// Mitsubishi GX Works2 project: 电路控制2   PLC: FX2N/FX2NC

PROGRAM MAIN
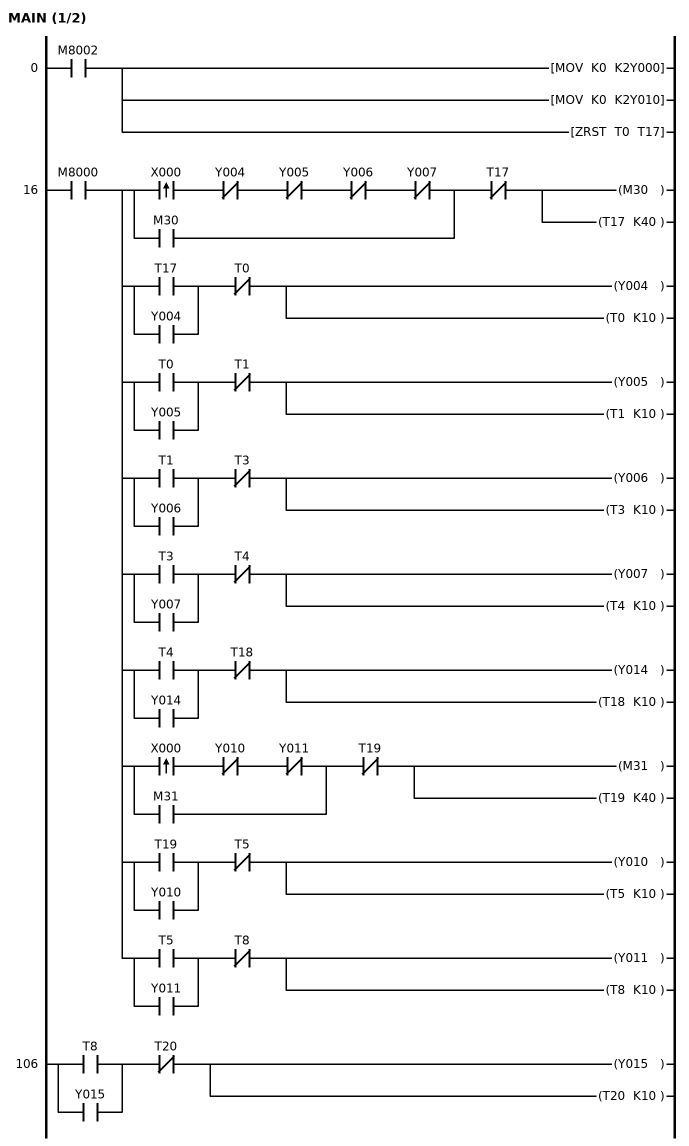
0     LD      M8002
      MOV     K0 K2Y000
      MOV     K0 K2Y010
      ZRST    T0 T17
16    LD      M8000
      MPS
      LDP     X000
      ANI     Y004
      ANI     Y005
      ANI     Y006
      ANI     Y007
      OR      M30
      ANB
      ANI     T17
      OUT     M30
      OUT     T17 K40
      MRD
      LD      T17
      OR      Y004
      ANB
      ANI     T0
      OUT     Y004
      OUT     T0 K10
      MRD
      LD      T0
      OR      Y005
      ANB
      ANI     T1
      OUT     Y005
      OUT     T1 K10
      MRD
      LD      T1
      OR      Y006
      ANB
      ANI     T3
      OUT     Y006
      OUT     T3 K10
      MRD
      LD      T3
      OR      Y007
      ANB
      ANI     T4
      OUT     Y007
      OUT     T4 K10
      MRD
      LD      T4
      OR      Y014
      ANB
      ANI     T18
      OUT     Y014
      OUT     T18 K10
      MRD
      LDP     X000
      ANI     Y010
      ANI     Y011
      OR      M31
      ANB
      ANI     T19
      OUT     M31
      OUT     T19 K40
      MRD
      LD      T19
      OR      Y010
      ANB
      ANI     T5
      OUT     Y010
      OUT     T5 K10
      MPP
      LD      T5
      OR      Y011
      ANB
      ANI     T8
      OUT     Y011
      OUT     T8 K10
106   LD      T8
      OR      Y015
      ANI     T20
      OUT     Y015
      OUT     T20 K10
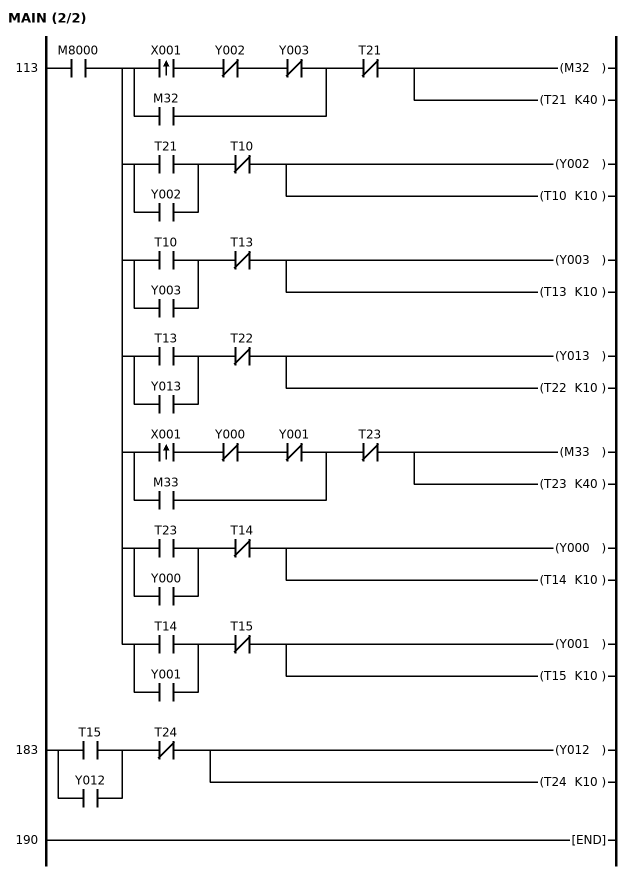
113   LD      M8000
      MPS
      LDP     X001
      ANI     Y002
      ANI     Y003
      OR      M32
      ANB
      ANI     T21
      OUT     M32
      OUT     T21 K40
      MRD
      LD      T21
      OR      Y002
      ANB
      ANI     T10
      OUT     Y002
      OUT     T10 K10
      MRD
      LD      T10
      OR      Y003
      ANB
      ANI     T13
      OUT     Y003
      OUT     T13 K10
      MRD
      LD      T13
      OR      Y013
      ANB
      ANI     T22
      OUT     Y013
      OUT     T22 K10
      MRD
      LDP     X001
      ANI     Y000
      ANI     Y001
      OR      M33
      ANB
      ANI     T23
      OUT     M33
      OUT     T23 K40
      MRD
      LD      T23
      OR      Y000
      ANB
      ANI     T14
      OUT     Y000
      OUT     T14 K10
      MPP
      LD      T14
      OR      Y001
      ANB
      ANI     T15
      OUT     Y001
      OUT     T15 K10
183   LD      T15
      OR      Y012
      ANI     T24
      OUT     Y012
      OUT     T24 K10
190   END
END_PROGRAM
